PROGRAM MAIN
VAR	
	//Test event
	stEvent : ST_Event;	
	bAddEvent : BOOL;
	CSVEventStorage : FB_CSVEventStorage;	
	fbEventLogger : FB_EventLogger(CSVEventStorage);
END_VAR

//Assign event values
stEvent.eEventType := E_Type.alarm;
stEvent.eEventSeverity := TCEventSeverity.Critical;
stEvent.nEventDefinition := 30;
stEvent.sEventMessage := 'Something went wrong';

//Run only once to add an event
IF bAddEvent THEN
	fbEventLogger.AddEvent(stEvent);
	bAddEvent := FALSE;
END_IF

END_PROGRAM

(* stored: Version 1.1.0.1, ProductVersion 3.1.4024.9
   POU MAIN: Id {efb1ca19-16d2-4253-8de9-e64b3dd80f65}, SpecialFunc None *)
